{attribute 'linkalways'} 
{attribute 'no_explicit_call' := 'This FB is a CLASS and must be accessed using methods or properties'}
{attribute 'enable_dynamic_creation'}
FUNCTION_BLOCK _ETcWatchdogAccumulationType EXTENDS EnumDatatypeBase
VAR
	localData : ETcWatchdogAccumulationType;
	activeData : REFERENCE TO ETcWatchdogAccumulationType;
	enumBaseDatatype : _UINT(localData);
END_VAR

METHOD PRIVATE AddLocalEnumeration
VAR_INPUT
	Enumeration : T_MAXSTRING;
	Value : ETcWatchdogAccumulationType;
END_VAR
AddEnumeration(Enumeration, Value);
END_METHOD

PROPERTY PUBLIC Address : PVOID
GET
Address := ADR(activeData);
END_GET
END_PROPERTY

METHOD PUBLIC ClearReference
VAR_INPUT
END_VAR
activeData REF= localData;
SetBaseDatatypeReference();
END_METHOD

METHOD PUBLIC Clone : I_Datatype
VAR
    pClone : POINTER TO _ETcWatchdogAccumulationType;
END_VAR
pClone := __NEW(_ETcWatchdogAccumulationType(InitialValue := Value));
Clone := pClone^;
END_METHOD

METHOD FB_init : BOOL
VAR_INPUT
	bInitRetains : BOOL; // if TRUE, the retain variables are initialized (warm start / cold start)
	bInCopyCode : BOOL;  // if TRUE, the instance afterwards gets moved into the copy code (online change)
	InitialValue : ETcWatchdogAccumulationType;
END_VAR
localData := InitialValue;
AddBaseDatatype(enumBaseDatatype);
ClearReference();

AddLocalEnumeration('WD_ACC_TYPE_MEAN', ETcWatchdogAccumulationType.WD_ACC_TYPE_MEAN);
AddLocalEnumeration('WD_ACC_TYPE_PRODUCT', ETcWatchdogAccumulationType.WD_ACC_TYPE_PRODUCT);
END_METHOD

PROPERTY PUBLIC Identifier : T_MAXSTRING
GET
Identifier := 'ETcWatchdogAccumulationType';
END_GET
END_PROPERTY

METHOD IsEnumeratorValueEqual : BOOL
VAR_INPUT
	Enumerator : I_KeyValueForwardEnumerator;
END_VAR
VAR
	storedValue : ETcWatchdogAccumulationType;
END_VAR
IF NOT Enumerator.TryGet(storedValue) THEN
	RETURN;
END_IF

IsEnumeratorValueEqual := storedValue = activeData;
END_METHOD

METHOD PUBLIC MakeReferenceTo
VAR_INPUT
	ReferenceTarget : REFERENCE TO ETcWatchdogAccumulationType;
END_VAR
activeData REF= ReferenceTarget;
SetBaseDatatypeReference();
END_METHOD

METHOD PROTECTED SetBaseDatatypeReference
VAR_INPUT
END_VAR
enumBaseDatatype.MakeReferenceTo(activeData);
END_METHOD

PROPERTY PUBLIC Size : UDINT
GET
Size := SIZEOF(activeData);
END_GET
END_PROPERTY

METHOD TryMakeReferenceTo : BOOL
VAR_INPUT
	Target : I_Datatype;
END_VAR
VAR
	targetAsEnum : I_EnumDatatype;
	pTargetData : POINTER TO ETcWatchdogAccumulationType;
END_VAR
IF NOT Target.TryResolveAsEnumDatatype(targetAsEnum) THEN
	RETURN;
END_IF

IF targetAsEnum.Identifier <> Identifier THEN
	RETURN;
END_IF

pTargetData := Target.Address;
activeData REF= pTargetData^;
SetBaseDatatypeReference();
TryMakeReferenceTo := TRUE;
END_METHOD

PROPERTY PUBLIC Value : ETcWatchdogAccumulationType
GET
Value := activeData;
END_GET
SET
activeData := Value;
END_SET
END_PROPERTY

END_FUNCTION_BLOCK

(* stored: Version 1.1.0.1, ProductVersion 3.1.4024.12
   POU _ETcWatchdogAccumulationType: Id {248d4af5-4761-03cb-3315-c6de778fc51d}, SpecialFunc None
   Folder Constructor: Id {9cf91514-1d0e-0c9f-1105-bf97c8986d40}
   Folder Private: Id {9d98cd08-4ecd-0ba2-1b23-e71709d12991}
   Folder Protected: Id {9cd420bd-0cba-0e35-1372-ae72c26a9279}
   Method AddLocalEnumeration: Id {bc0316d8-c303-020f-3200-ae372d69f243}
   Property Address: Id {a420a4cc-0b4e-0578-2a44-f6b806f8a472}
   Get Get: Id {fc6a92d7-1cd5-0fb9-2f67-a7e22c39139a}
   Method ClearReference: Id {93be8b33-bff7-0c63-1ebf-ecc7fde8b977}
   Method Clone: Id {d783b119-eac7-08e7-1495-114df27e59f8}
   Method FB_init: Id {d84dcc2b-0aea-0310-3881-9d4ecee4af73}
   Property Identifier: Id {b4fd7588-94ae-05a9-0ccf-0ddee244e725}
   Get Get: Id {9d30c0f5-c52f-0a9d-395d-3bb1ee02809c}
   Method IsEnumeratorValueEqual: Id {4b28fff7-d5fa-0a61-3439-5b0d680ba79c}
   Method MakeReferenceTo: Id {d506d6b7-08c5-0f86-3479-5c7517ffa7bf}
   Method SetBaseDatatypeReference: Id {5dbd722c-45c3-0735-3b0e-3cb537a4e155}
   Property Size: Id {a2e20e97-fc60-0212-1c11-dad838975655}
   Get Get: Id {07011bde-818a-031b-0f6e-d496f516f370}
   Method TryMakeReferenceTo: Id {a9b2d746-b49f-005d-3840-698b7489c635}
   Property Value: Id {8fa63e82-dca6-0213-0e07-7175b061756a}
   Get Get: Id {12f7bc20-aae5-0064-309b-30475507dcf4}
   Set Set: Id {37328d45-9662-00c1-18d4-b13c7c17457c} *)
